% RSLogix 500 project I2P Hands On Test 1 - Daniel.RSS, saved by version 10.00.00.00 %
PROJECT "UNTITLED"    % processor: Bul.1763 MicroLogix 1100 Series B %

PROGRAM FILES
  LAD 2   6 rungs

DATA FILES
  O0 OUTPUT  4 elements
  I1 INPUT  6 elements
  S2 STATUS  66 elements
  B3 BINARY  1 elements
  T4 TIMER  1 elements
  C5 COUNTER  1 elements
  R6 CONTROL  1 elements
  N7 INTEGER  1 elements
  F8 FLOAT  1 elements

LADDER 2
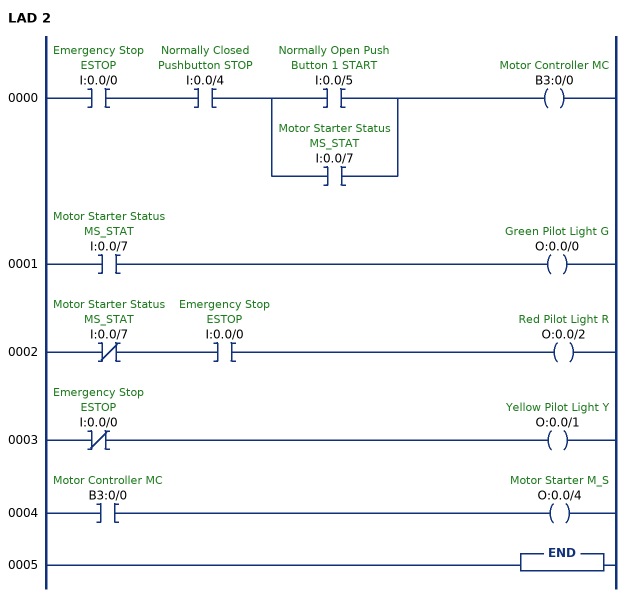
% Rung: 0 %
SOR XIC I:0.0/0 XIC I:0.0/4 BST XIC I:0.0/5 NXB XIC I:0.0/7 BND OTE B3:0/0 EOR
%   I:0.0/0  ESTOP  "Emergency Stop" %
%   I:0.0/4  STOP  "Normally Closed Pushbutton" %
%   I:0.0/5  START  "Normally Open Push Button 1" %
%   I:0.0/7  MS_STAT  "Motor Starter Status" %
%   B3:0/0  MC  "Motor Controller" %
% Rung: 1 %
SOR XIC I:0.0/7 OTE O:0.0/0 EOR
%   I:0.0/7  MS_STAT  "Motor Starter Status" %
%   O:0.0/0  G  "Green Pilot Light" %
% Rung: 2 %
SOR XIO I:0.0/7 XIC I:0.0/0 OTE O:0.0/2 EOR
%   I:0.0/7  MS_STAT  "Motor Starter Status" %
%   I:0.0/0  ESTOP  "Emergency Stop" %
%   O:0.0/2  R  "Red Pilot Light" %
% Rung: 3 %
SOR XIO I:0.0/0 OTE O:0.0/1 EOR
%   I:0.0/0  ESTOP  "Emergency Stop" %
%   O:0.0/1  Y  "Yellow Pilot Light" %
% Rung: 4 %
SOR XIC B3:0/0 OTE O:0.0/4 EOR
%   B3:0/0  MC  "Motor Controller" %
%   O:0.0/4  M_S  "Motor Starter" %
% Rung: 5 %
SOR END EOR

OTHER DOCUMENTED ADDRESSES
  I:0.0/1  3PSSA  "Three Position Selector Switch Position A"
  I:0.0/2  3PSSB  "Three Position Selector Switch Position B"
  I:0.0/3  2PSS  "Two Position Selector Switch"
  I:0.0/6  NOPB2  "Normally Open Push Button 2"
  I:0.0/8  MSF  "Motor Starter Forward"
  I:0.0/9  MSR  "Motor Starter Reverse"
  O:0.0/3  B  "Blue Pilot Light"
  O:0.0/5  MS  "Motor Starter"
